TYPE ZCom :
STRUCT
  // module context
  App : ZApplication.ApplicationComPublish;
  Alarming : ZApplication.AlarmingCom;
  Messages : ZApplication.MessagingCom;
  
  // unit context
  Unit : ZComUnit;

END_STRUCT
END_TYPE

(* stored: Version 1.1.0.1
   DUT ZCom: Id {9ecb853e-df32-4f3b-a2df-b7078a62f6ec} *)
